FUNCTION_BLOCK Zone EXTENDS Objective
VAR

    internalStartPosition : LREAL;
    internalEndPosition   : LREAL;
	internalTrack : REFERENCE TO Track; 

    internalMoverList : MoverList;

END_VAR

{attribute 'monitoring' := 'call'}
PROPERTY CurrentMoverCount : USINT
GET
CurrentMoverCount := THIS^.CurrentMoverList.TrackedMoverCount;
END_GET
END_PROPERTY

PROPERTY CurrentMoverList : iMoverList
GET
VAR
    i : ulint;
	moverTrackId: INT;
END_VAR
internalMoverList.UnregisterAll();

FOR i := 1 TO SIZEOF(TrackedMovers) / SIZEOF(internalTrackedMovers[1]) DO
    IF internalTrackedMovers[i] <> 0 AND_THEN internalTrackedMovers[i]^.IsTrackReady AND internalTrackedMovers[i]^.CurrentTrack <> 0 THEN
		moverTrackId := internalTrackedMovers[i]^.CurrentTrack^.Id;
		IF (moverTrackId = internalTrack.Id) THEN
			IF internalStartPosition < internalEndPosition
				   AND internalTrackedMovers[i]^.TrackInfo.TrackPosition > internalStartPosition
				   AND internalTrackedMovers[i]^.TrackInfo.TrackPosition < internalEndPosition THEN
				// Zone does NOT contain the rollover point, and DOES contain the mover
	
				internalMoverList.RegisterMover(internalTrackedMovers[i]^);
	
			ELSIF internalStartPosition > internalEndPosition
					  AND (internalTrackedMovers[i]^.TrackInfo.TrackPosition > internalStartPosition
					  OR internalTrackedMovers[i]^.TrackInfo.TrackPosition < internalEndPosition) THEN
				// Zone DOES contain the rollover point, and DOES contain the mover
	
				internalMoverList.RegisterMover(internalTrackedMovers[i]^);
	
			ELSE
				// Either the zone doesn't contain this mover,
				// Or the StartPosition and EndPosition are coincident. Either way, add no movers
			END_IF
		END_IF
    END_IF
END_FOR

CurrentMoverList := internalMoverList;
END_GET
END_PROPERTY

{attribute 'monitoring' := 'call'}
PROPERTY EndPosition : LREAL
GET
EndPosition := internalEndPosition;
END_GET
SET
// todo add limit checks?
internalEndPosition := EndPosition;
END_SET
END_PROPERTY

METHOD GetMover : REFERENCE TO Mover
VAR_INPUT
    Index     : USINT;                // 0 is find the first closest mover, 1 is find the second closest mover, 2 is find the third, etc. etc. etc.
    Direction : Tc2_MC2.MC_Direction; // Positive = find the mover closest to the End Position. Negative = find the mover closest to the Start Position
END_VAR



IF Direction = MC_Positive_Direction THEN
    GetMover REF= THIS^.CurrentMoverList.GetMoverByLocation(Index, THIS^.EndPosition, MC_Positive_Direction);
	GetMover.SourceInstancePath		:= THIS^.InstancePath;
ELSIF Direction = MC_Negative_Direction THEN
    GetMover REF= THIS^.CurrentMoverList.GetMoverByLocation(Index, THIS^.StartPosition, MC_Negative_Direction);
	GetMover.SourceInstancePath		:= THIS^.InstancePath;
ELSE
    GetMover REF= 0;
END_IF

// If the Zone has no mover to return given the input parameters, then return an imposter ErrorMover
IF __ISVALIDREF(GetMover) = FALSE THEN
	ErrorMover.SourceInstancePath	:= THIS^.InstancePath;
	GetMover						REF= ErrorMover;
END_IF
END_METHOD

METHOD SetTrack : BOOL
VAR_INPUT
	Track : REFERENCE TO TRACK;
END_VAR
internalTrack REF= Track;
END_METHOD

{attribute 'monitoring' := 'call'}
PROPERTY StartPosition : LREAL
GET
StartPosition := internalStartPosition;
END_GET
SET
// Todo add limit checks?
internalStartPosition := StartPosition;
END_SET
END_PROPERTY

PROPERTY TrackId : DINT
GET
TrackId := internalTrack.Id;
END_GET
END_PROPERTY

{attribute 'monitoring' := 'call'}
PROPERTY ZoneLength : LREAL
GET
IF internalStartPosition < internalEndPosition THEN
    // Zone does NOT include the rollover point
    ZoneLength := internalEndPosition - internalStartPosition;
ELSIF internalStartPosition > internalEndPosition THEN
    // Zone DOES include the rollover point
    ZoneLength := internalEndPosition + (internalEndPosition + internalTrack.Length - internalStartPosition);
ELSE
    // Start and end position are coincident, ZL is 0
    ZoneLength := 0;
END_IF
END_GET
END_PROPERTY

END_FUNCTION_BLOCK

(* stored: Version 1.1.0.1, ProductVersion 3.1.4026.8
   POU Zone: Id {de9b5dde-c203-4f4d-abe0-431568995536}, SpecialFunc None
   Folder Methods: Id {c12d9132-64a8-40b2-b1d9-3d115c20d531}
   Folder Properties: Id {90c52b3d-9a13-4439-896a-3c5f735e1216}
   Property CurrentMoverCount: Id {2570f0bb-44d6-0dc6-396c-15aba6800423}
   Get Get: Id {6103a49f-65cc-06b3-2883-ee1cd1651525}
   Property CurrentMoverList: Id {fba40b8e-82e6-48ba-a30f-3cc9abb7a1fc}
   Get Get: Id {9681b7d1-44db-47ce-812f-f41b5199fc2d}
   Property EndPosition: Id {0a5f097e-96c3-43a1-b536-04f368f24ca3}
   Get Get: Id {a512e404-14bd-4b1c-9731-3bba7de351df}
   Set Set: Id {5303700b-9c9b-41e5-8b19-d6050a760e26}
   Method GetMover: Id {faabc650-b1f1-4ef7-8da9-de80f9ce94fc}
   Method SetTrack: Id {7cc8b098-587a-05e2-14ee-fd833da9898e}
   Property StartPosition: Id {aacc7e02-3b0c-44c1-b85c-a6193164623c}
   Get Get: Id {3c066f4a-ee41-4a60-96e5-d5b56be91452}
   Set Set: Id {c038cebd-9252-42ab-8a7b-34fa884ebed1}
   Property TrackId: Id {fa238337-4029-0a7e-0a02-4f8a1ea15d7d}
   Get Get: Id {2dbe3079-85d1-0042-009b-dd035bd899ff}
   Property ZoneLength: Id {cc1fdc68-29d3-4f91-948b-3fe78f7d05d8}
   Get Get: Id {6d92c621-884a-4d2c-8ab0-83911c1e9108} *)
